INTERFACE I_XtsSystemNctManager EXTENDS I_Base, I_XtsTask, XtsCore.I_Cyclic

PROPERTY NctController : I_TcIoXtsNctController
GET
END_GET
END_PROPERTY

END_INTERFACE

(* stored: Version 1.1.0.1, ProductVersion 3.1.4026.19
   Itf I_XtsSystemNctManager: Id {804ddc44-c73c-4877-90a2-51374a429fbd}
   Property NctController: Id {af7ad85a-ff70-48dd-a662-0b0355854eea}
   Get Get: Id {3133fdf4-4bb9-44f6-8097-f7c1051686ed} *)
